RoboDK station: container_v08_small.rdk

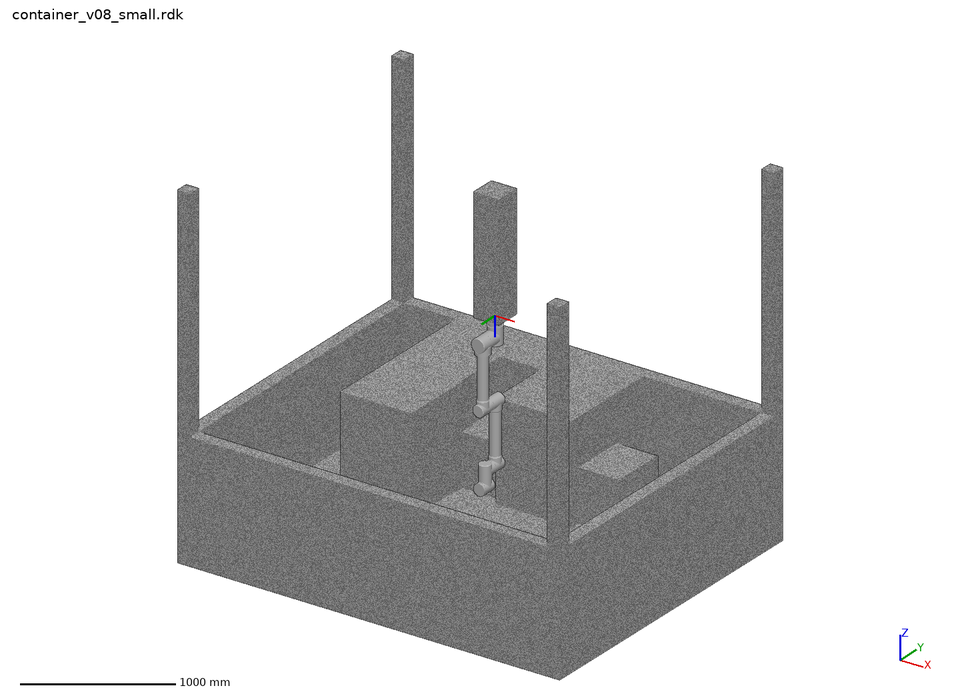
[picture v0: the station drawn from its stored meshes, robots at their saved joint values, targets as dots, program paths as lines]
Station container_v08_small (saved by RoboDK 5.4.0). Poses are relative to the parent item; angles as X-Y-Z fixed-axis rotations.
  - object kontener v08 stp at (0, 0, 0) mm, size 3000 x 2500 x 2665 mm, geometry from kontener v08 stp.stp
  - frame avena_arm Base at (607.5, -10, 1600) mm, rotated rx 180 ry 0 rz 0 deg
    - robot avena_arm: 6 axes
        modified DH rows (alpha deg, a mm, theta deg, d mm): 0, 0, 0, 139.3; 90, 0, 90, 0; 0, 467, 0, 0; 0, 452, -90, -113.5; -90, 0, 180, 113.5; 90, 0, 0, 68.1
        joint limits [-174.8, -90, -166.2, -174.8, -174.8, -174.8] to [174.8, 90, 166.2, 174.8, 174.8, 174.8]; home [0, 0, 0, 0, 0, 0]; saved at [0, 0, 0, 0, 0, 0]
